// Mitsubishi GX Works2 project: Smart Geezer   PLC: FX3G

PROGRAM MAIN
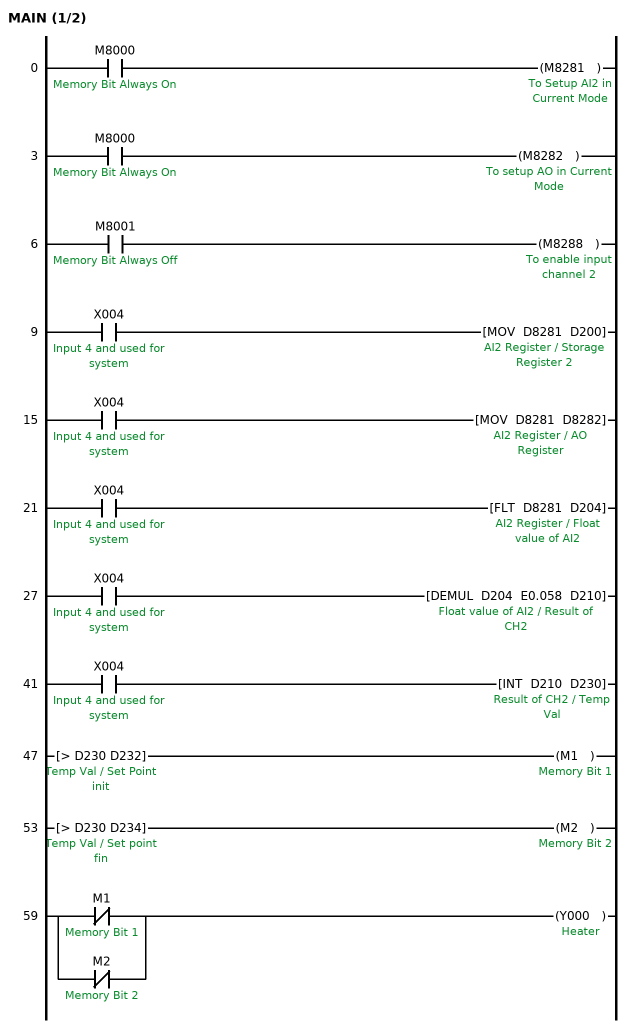
0     LD      M8000  ; Memory Bit Always On
      OUT     M8281  ; To Setup AI2 in Current Mode
3     LD      M8000  ; Memory Bit Always On
      OUT     M8282  ; To setup AO in Current Mode
6     LD      M8001  ; Memory Bit Always Off
      OUT     M8288  ; To enable input channel 2
9     LD      X004  ; Input 4 and used for system
      MOV     D8281 D200  ; AI2 Register / Storage Register 2
15    LD      X004  ; Input 4 and used for system
      MOV     D8281 D8282  ; AO Register
21    LD      X004  ; Input 4 and used for system
      FLT     D8281 D204  ; Float value of AI2
27    LD      X004  ; Input 4 and used for system
      DEMUL   D204 E0.058 D210  ; Result of CH2
41    LD      X004  ; Input 4 and used for system
      INT     D210 D230  ; Temp Val
47    LD>     D230 D232  ; Temp Val / Set Point init
      OUT     M1  ; Memory Bit 1
53    LD>     D230 D234  ; Temp Val / Set point fin
      OUT     M2  ; Memory Bit 2
59    LDI     M1  ; Memory Bit 1
      ORI     M2  ; Memory Bit 2
      OUT     Y000  ; Heater
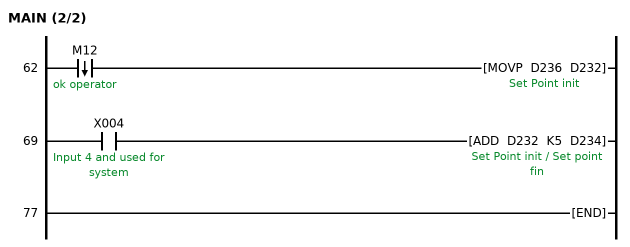
62    LDF     M12  ; ok operator
      MOVP    D236 D232
69    LD      X004  ; Input 4 and used for system
      ADD     D232 K5 D234
77    END
END_PROGRAM

// device comments not shown above
M0  ; Memory bit 0
M3  ; Memory Bit 3
M4  ; Memory Bit 4
M10  ; increment operator
M11  ; decrement operator
D0  ; Data register for setpoint
D100  ; Storage Register 1
D104  ; Float value of AI1
D106  ; Initial Value of AI1
D108  ; Resulted Value
D110  ; Result of CH1
D112  ; Final value of AI1
D120  ; CH1 final result
D130  ; Int of ch1
D132  ; Temp Const
D134  ; Temp Const
D206  ; Initial value of AI2
D208  ; Resulted value
D212  ; Final value of AI2
D220  ; CH2 final value
T0  ; timer0 with 100ms delay
T1  ; timer1 with 100ms delay
